// Mitsubishi GX Works2 project: SmartFarmModbusTempDx   PLC: FX3U/FX3UC

PROGRAM MAIN
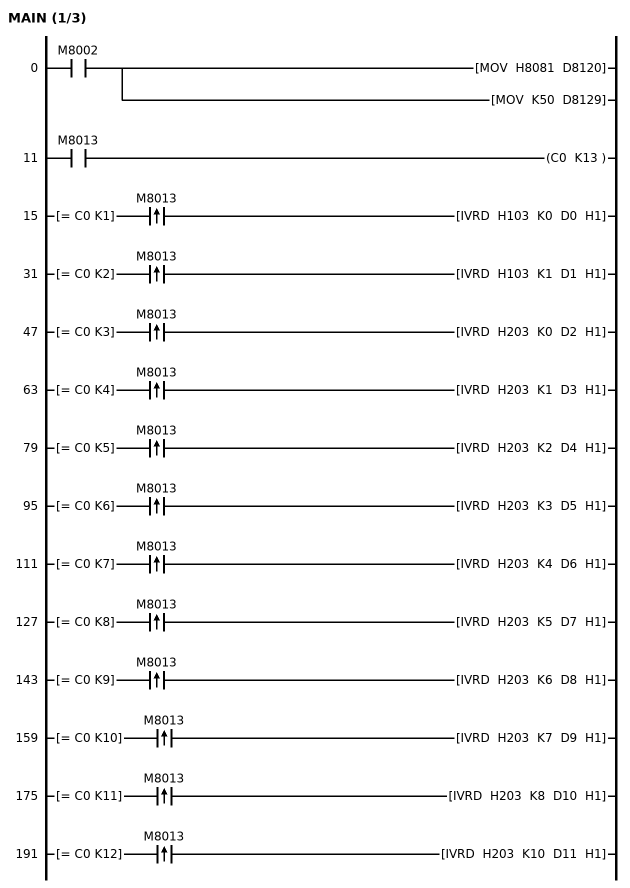
0     LD      M8002
      MOV     H8081 D8120
      MOV     K50 D8129
11    LD      M8013
      OUT     C0 K13
15    LD=     C0 K1
      ANDP    M8013
      IVRD    H103 K0 D0 H1
31    LD=     C0 K2
      ANDP    M8013
      IVRD    H103 K1 D1 H1
47    LD=     C0 K3
      ANDP    M8013
      IVRD    H203 K0 D2 H1
63    LD=     C0 K4
      ANDP    M8013
      IVRD    H203 K1 D3 H1
79    LD=     C0 K5
      ANDP    M8013
      IVRD    H203 K2 D4 H1
95    LD=     C0 K6
      ANDP    M8013
      IVRD    H203 K3 D5 H1
111   LD=     C0 K7
      ANDP    M8013
      IVRD    H203 K4 D6 H1
127   LD=     C0 K8
      ANDP    M8013
      IVRD    H203 K5 D7 H1
143   LD=     C0 K9
      ANDP    M8013
      IVRD    H203 K6 D8 H1
159   LD=     C0 K10
      ANDP    M8013
      IVRD    H203 K7 D9 H1
175   LD=     C0 K11
      ANDP    M8013
      IVRD    H203 K8 D10 H1
191   LD=     C0 K12
      ANDP    M8013
      IVRD    H203 K10 D11 H1
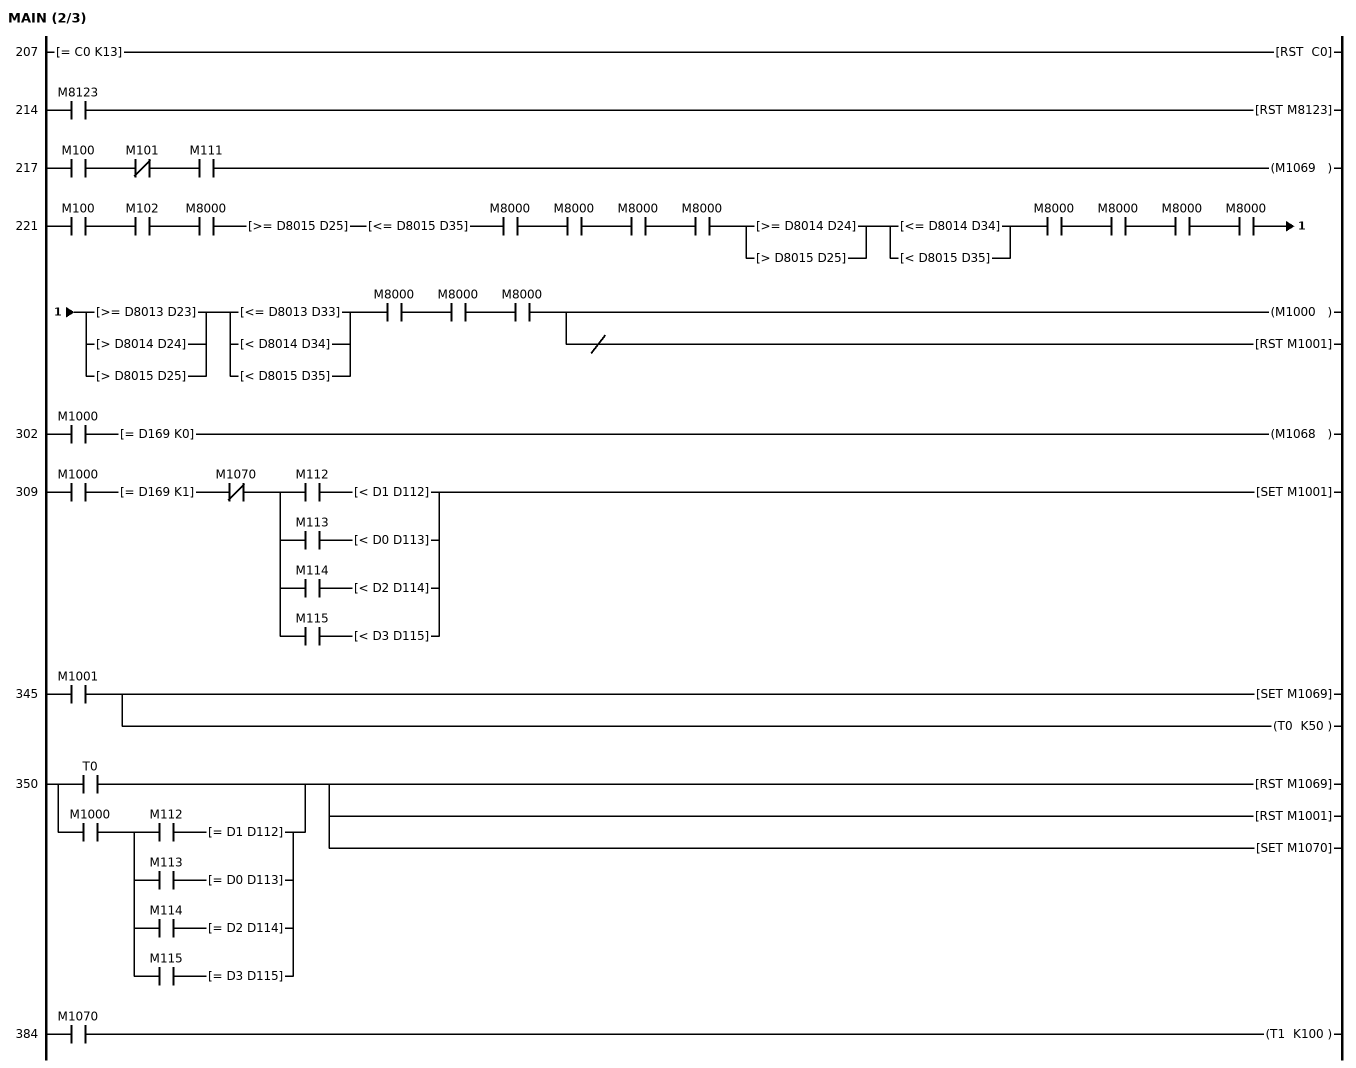
207   LD=     C0 K13
      RST     C0
214   LD      M8123
      RST     M8123
217   LD      M100
      ANI     M101
      AND     M111
      OUT     M1069
221   LD      M100
      AND     M102
      AND     M8000
      AND>=   D8015 D25
      AND<=   D8015 D35
      AND     M8000
      AND     M8000
      AND     M8000
      AND     M8000
      LD>=    D8014 D24
      OR>     D8015 D25
      ANB
      LD<=    D8014 D34
      OR<     D8015 D35
      ANB
      AND     M8000
      AND     M8000
      AND     M8000
      AND     M8000
      LD>=    D8013 D23
      OR>     D8014 D24
      OR>     D8015 D25
      ANB
      LD<=    D8013 D33
      OR<     D8014 D34
      OR<     D8015 D35
      ANB
      AND     M8000
      AND     M8000
      AND     M8000
      OUT     M1000
      INV
      RST     M1001
302   LD      M1000
      AND=    D169 K0
      OUT     M1068
309   LD      M1000
      AND=    D169 K1
      ANI     M1070
      LD      M112
      AND<    D1 D112
      LD      M113
      AND<    D0 D113
      ORB
      LD      M114
      AND<    D2 D114
      ORB
      LD      M115
      AND<    D3 D115
      ORB
      ANB
      SET     M1001
345   LD      M1001
      SET     M1069
      OUT     T0 K50
350   LD      T0
      LD      M1000
      LD      M112
      AND=    D1 D112
      LD      M113
      AND=    D0 D113
      ORB
      LD      M114
      AND=    D2 D114
      ORB
      LD      M115
      AND=    D3 D115
      ORB
      ANB
      ORB
      RST     M1069
      RST     M1001
      SET     M1070
384   LD      M1070
      OUT     T1 K100
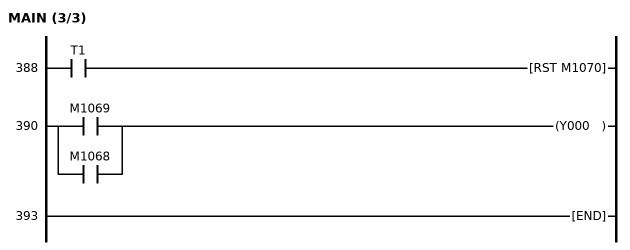
388   LD      T1
      RST     M1070
390   LD      M1069
      OR      M1068
      OUT     Y000
393   END
END_PROGRAM
